FUNCTION_BLOCK E_Split16 (* Composite Function Block Type *)
  (* Standard: 61499-2 *)
  (* Version 0.0, 2018-12-21, 4DIAC-IDE, 4DIAC-Consortium *)
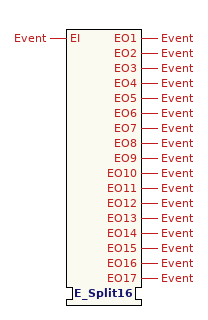
  EVENT_INPUT
    EI;
  END_EVENT
  EVENT_OUTPUT
    EO1;
    EO2;
    EO3;
    EO4;
    EO5;
    EO6;
    EO7;
    EO8;
    EO9;
    EO10;
    EO11;
    EO12;
    EO13;
    EO14;
    EO15;
    EO16;
    EO17;
  END_EVENT
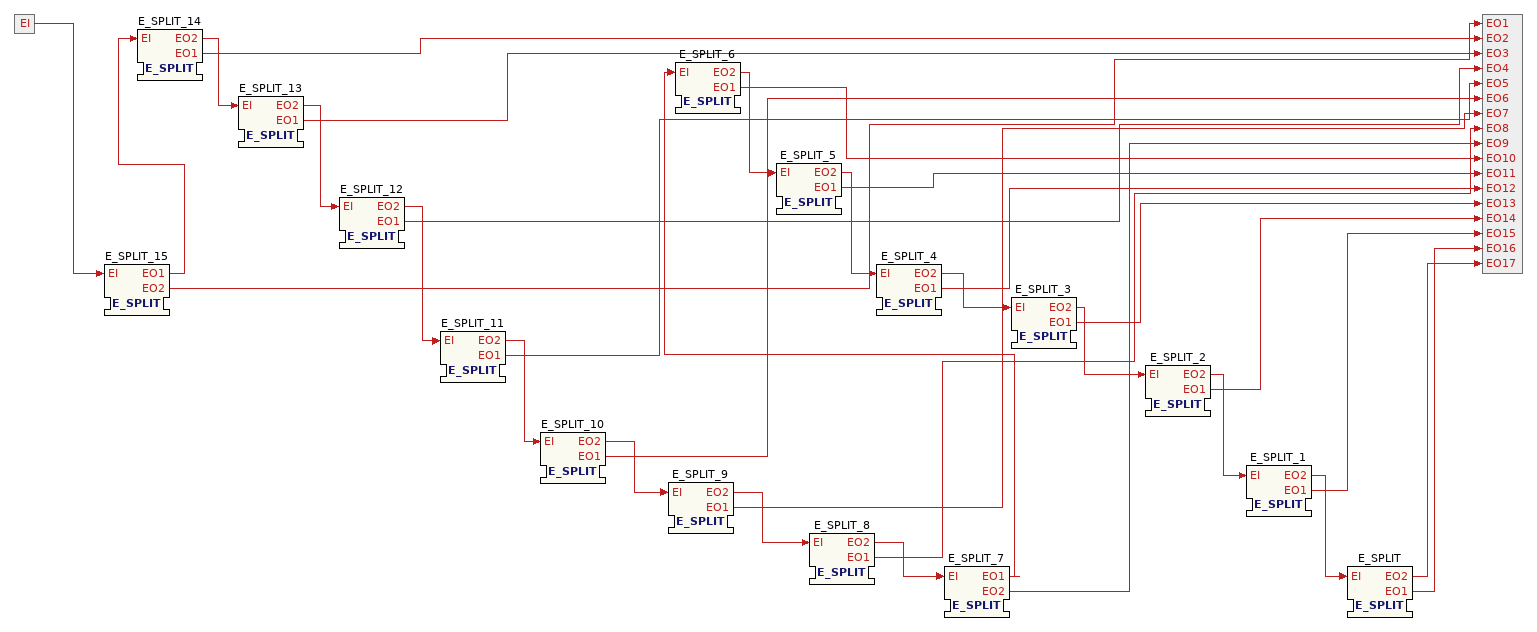
  FBS
    E_SPLIT : E_SPLIT;
    E_SPLIT_1 : E_SPLIT;
    E_SPLIT_2 : E_SPLIT;
    E_SPLIT_3 : E_SPLIT;
    E_SPLIT_4 : E_SPLIT;
    E_SPLIT_5 : E_SPLIT;
    E_SPLIT_6 : E_SPLIT;
    E_SPLIT_7 : E_SPLIT;
    E_SPLIT_8 : E_SPLIT;
    E_SPLIT_9 : E_SPLIT;
    E_SPLIT_10 : E_SPLIT;
    E_SPLIT_11 : E_SPLIT;
    E_SPLIT_12 : E_SPLIT;
    E_SPLIT_13 : E_SPLIT;
    E_SPLIT_14 : E_SPLIT;
    E_SPLIT_15 : E_SPLIT;
  END_FBS
  EVENT_CONNECTIONS
    E_SPLIT.EO2 TO EO17;
    E_SPLIT.EO1 TO EO16;
    E_SPLIT_1.EO2 TO E_SPLIT.EI;
    E_SPLIT_1.EO1 TO EO15;
    E_SPLIT_2.EO2 TO E_SPLIT_1.EI;
    E_SPLIT_2.EO1 TO EO14;
    E_SPLIT_3.EO2 TO E_SPLIT_2.EI;
    E_SPLIT_3.EO1 TO EO13;
    E_SPLIT_4.EO2 TO E_SPLIT_3.EI;
    E_SPLIT_4.EO1 TO EO12;
    E_SPLIT_5.EO2 TO E_SPLIT_4.EI;
    E_SPLIT_5.EO1 TO EO11;
    E_SPLIT_6.EO2 TO E_SPLIT_5.EI;
    E_SPLIT_6.EO1 TO EO10;
    E_SPLIT_7.EO1 TO E_SPLIT_6.EI;
    E_SPLIT_7.EO2 TO EO9;
    E_SPLIT_8.EO2 TO E_SPLIT_7.EI;
    E_SPLIT_8.EO1 TO EO8;
    E_SPLIT_9.EO2 TO E_SPLIT_8.EI;
    E_SPLIT_9.EO1 TO EO7;
    E_SPLIT_10.EO2 TO E_SPLIT_9.EI;
    E_SPLIT_10.EO1 TO EO6;
    E_SPLIT_11.EO2 TO E_SPLIT_10.EI;
    E_SPLIT_11.EO1 TO EO5;
    E_SPLIT_12.EO2 TO E_SPLIT_11.EI;
    E_SPLIT_12.EO1 TO EO4;
    E_SPLIT_13.EO2 TO E_SPLIT_12.EI;
    E_SPLIT_13.EO1 TO EO3;
    E_SPLIT_14.EO2 TO E_SPLIT_13.EI;
    E_SPLIT_14.EO1 TO EO2;
    E_SPLIT_15.EO1 TO E_SPLIT_14.EI;
    E_SPLIT_15.EO2 TO EO1;
    EI TO E_SPLIT_15.EI;
  END_CONNECTIONS
END_FUNCTION_BLOCK
